TYPE json_st :
STRUCT
	{attribute 'json' := 'name'}
	name : STRING;
	{attribute 'json' := 'age'}
	age : INT;
	{attribute 'json' := 'car'}
	car : STRING;
END_STRUCT
END_TYPE

(* stored: Version 1.1.0.1, ProductVersion 3.1.4024.4
   DUT json_st: Id {57d9c0de-990c-435b-b176-07fd3b3060ca} *)
